// TIA Portal V17 export
// export: Created 2025-03-05T08:00:56.7108136Z, ExportSetting WithDefaults, DisplayName Totally Integrated Automation Portal, DisplayVersion V17 Update 8, DisplayName TIA Portal Openness, DisplayVersion V17 Update 8, DisplayName TIA Portal Version Control Interface, DisplayVersion V17, DisplayName SINAMICS Startdrive Advanced, DisplayVersion V17 SP2, DisplayName SINAMICS Startdrive G110M, G120, G120C, G120D, G120P, G115D, DisplayVersion V17 SP2, DisplayName SINAMICS Startdrive G130, G150, S120, S150, SINAMICS MV, S210, DisplayVersion V17 SP2, DisplayName STEP 7 Professional, DisplayVersion V17 Update 8, DisplayName SINUMERIK ONE STEP 7 Toolbox, DisplayVersion V17 Update 12, DisplayName SINUMERIK 840D sl STEP 7 Toolbox, DisplayVersion V17 Update 12, DisplayName STEP 7 Safety, DisplayVersion V17 Update 6, DisplayName WinCC Advanced, DisplayVersion V17 Update 8
FUNCTION "FC1502_PROTECTION_GAS" : Void   // FC1502, LAD
{ S7_Optimized_Access := 'TRUE' }
VERSION : 0.1
// stored: AutoNumber false, IsIECCheckEnabled false, SetENOAutomatically false, UDAEnableTagReadback false
   VAR_TEMP
      GAS_FLOW_TEMP_AUX : Real;
   END_VAR
BEGIN

REGION Network 1: PROTECTION GAS VALVE UNIT 01
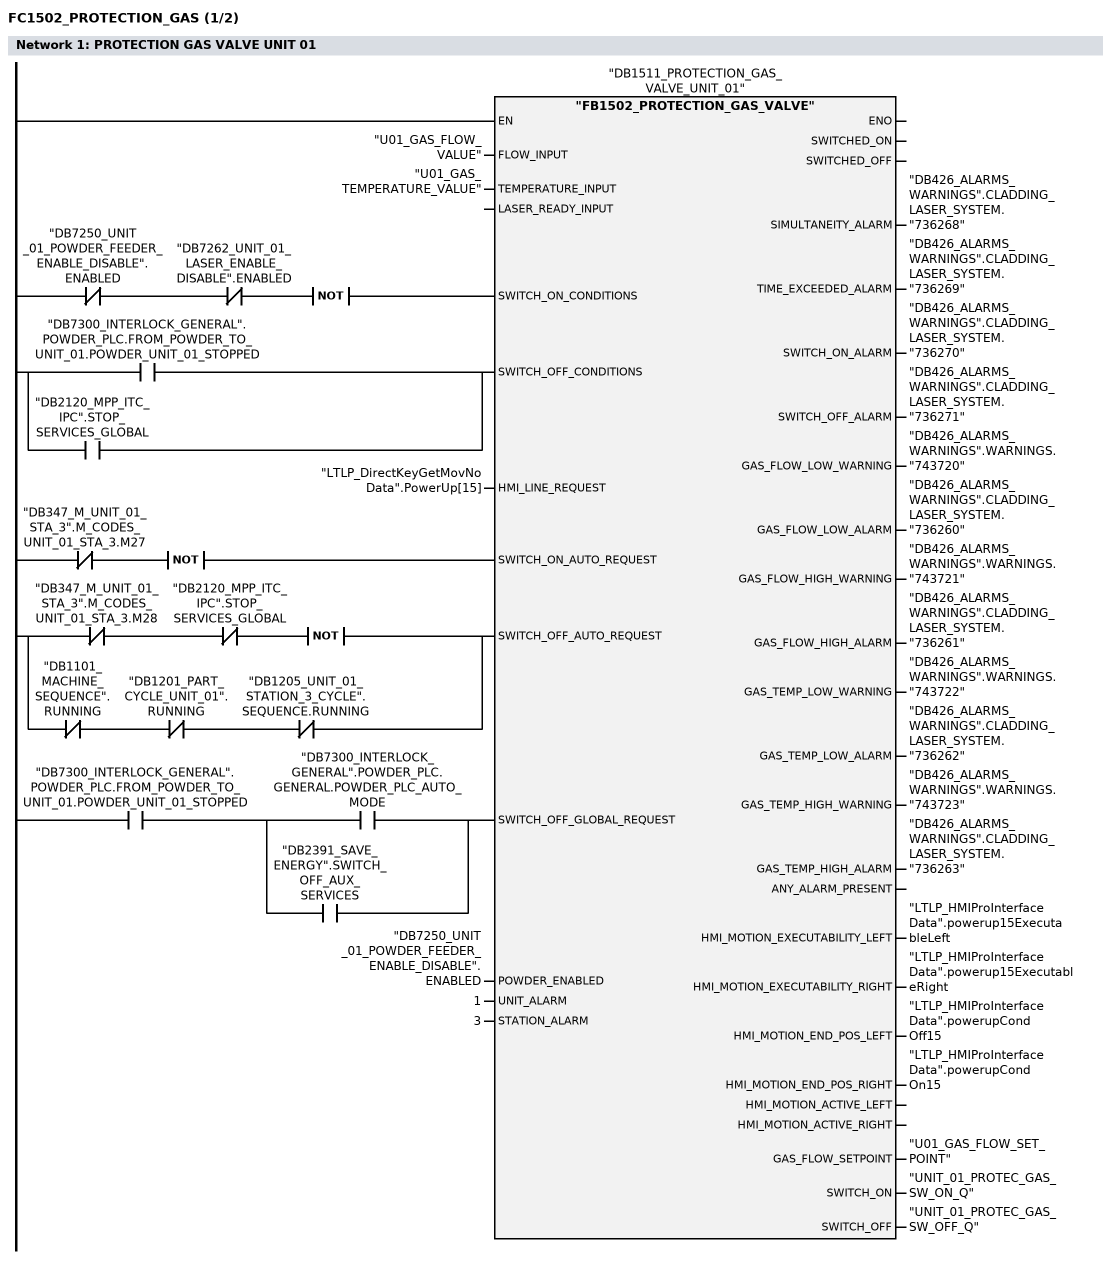
   RUNG wire#powerrail
      "DB1511_PROTECTION_GAS_VALVE_UNIT_01"(SWITCH_ON_CONDITIONS := wire#w1, SWITCH_OFF_CONDITIONS := wire#w2, SWITCH_ON_AUTO_REQUEST := wire#w3, SWITCH_OFF_AUTO_REQUEST := wire#w4, SWITCH_OFF_GLOBAL_REQUEST := wire#w6, FLOW_INPUT := "U01_GAS_FLOW_VALUE", TEMPERATURE_INPUT := "U01_GAS_TEMPERATURE_VALUE", LASER_READY_INPUT :=, HMI_LINE_REQUEST := "LTLP_DirectKeyGetMovNoData".PowerUp[15], POWDER_ENABLED := "DB7250_UNIT _01_POWDER_FEEDER_ENABLE_DISABLE".ENABLED, UNIT_ALARM := 1, STATION_ALARM := 3, SWITCHED_ON =>, SWITCHED_OFF =>, SIMULTANEITY_ALARM => "DB426_ALARMS_WARNINGS".CLADDING_LASER_SYSTEM."736268", TIME_EXCEEDED_ALARM => "DB426_ALARMS_WARNINGS".CLADDING_LASER_SYSTEM."736269", SWITCH_ON_ALARM => "DB426_ALARMS_WARNINGS".CLADDING_LASER_SYSTEM."736270", SWITCH_OFF_ALARM => "DB426_ALARMS_WARNINGS".CLADDING_LASER_SYSTEM."736271", GAS_FLOW_LOW_WARNING => "DB426_ALARMS_WARNINGS".WARNINGS."743720", GAS_FLOW_LOW_ALARM => "DB426_ALARMS_WARNINGS".CLADDING_LASER_SYSTEM."736260", GAS_FLOW_HIGH_WARNING => "DB426_ALARMS_WARNINGS".WARNINGS."743721", GAS_FLOW_HIGH_ALARM => "DB426_ALARMS_WARNINGS".CLADDING_LASER_SYSTEM."736261", GAS_TEMP_LOW_WARNING => "DB426_ALARMS_WARNINGS".WARNINGS."743722", GAS_TEMP_LOW_ALARM => "DB426_ALARMS_WARNINGS".CLADDING_LASER_SYSTEM."736262", GAS_TEMP_HIGH_WARNING => "DB426_ALARMS_WARNINGS".WARNINGS."743723", GAS_TEMP_HIGH_ALARM => "DB426_ALARMS_WARNINGS".CLADDING_LASER_SYSTEM."736263", ANY_ALARM_PRESENT =>, HMI_MOTION_EXECUTABILITY_LEFT => "LTLP_HMIProInterfaceData".powerup15ExecutableLeft, HMI_MOTION_EXECUTABILITY_RIGHT => "LTLP_HMIProInterfaceData".powerup15ExecutableRight, HMI_MOTION_END_POS_LEFT => "LTLP_HMIProInterfaceData".powerupCondOff15, HMI_MOTION_END_POS_RIGHT => "LTLP_HMIProInterfaceData".powerupCondOn15, HMI_MOTION_ACTIVE_LEFT =>, HMI_MOTION_ACTIVE_RIGHT =>, GAS_FLOW_SETPOINT => "U01_GAS_FLOW_SET_POINT", SWITCH_ON => "UNIT_01_PROTEC_GAS_SW_ON_Q", SWITCH_OFF => "UNIT_01_PROTEC_GAS_SW_OFF_Q")
   END_RUNG
   RUNG wire#powerrail
      I_Contact( "DB7250_UNIT _01_POWDER_FEEDER_ENABLE_DISABLE".ENABLED )
      I_Contact( "DB7262_UNIT_01_LASER_ENABLE_DISABLE".ENABLED )
      Not()
   END_RUNG wire#w1
   RUNG wire#powerrail
      Contact( "DB7300_INTERLOCK_GENERAL".POWDER_PLC.FROM_POWDER_TO_UNIT_01.POWDER_UNIT_01_STOPPED )
   END_RUNG wire#w2
   RUNG wire#powerrail
      Contact( "DB2120_MPP_ITC_IPC".STOP_SERVICES_GLOBAL )
   END_RUNG wire#w2
   RUNG wire#powerrail
      I_Contact( "DB347_M_UNIT_01_STA_3".M_CODES_UNIT_01_STA_3.M27 )
      Not()
   END_RUNG wire#w3
   RUNG wire#powerrail
      I_Contact( "DB347_M_UNIT_01_STA_3".M_CODES_UNIT_01_STA_3.M28 )
      I_Contact( "DB2120_MPP_ITC_IPC".STOP_SERVICES_GLOBAL )
      Not()
   END_RUNG wire#w4
   RUNG wire#powerrail
      I_Contact( "DB1101_MACHINE_SEQUENCE".RUNNING )
      I_Contact( "DB1201_PART_CYCLE_UNIT_01".RUNNING )
      I_Contact( "DB1205_UNIT_01_STATION_3_CYCLE".SEQUENCE.RUNNING )
   END_RUNG wire#w4
   RUNG wire#powerrail
      Contact( "DB7300_INTERLOCK_GENERAL".POWDER_PLC.FROM_POWDER_TO_UNIT_01.POWDER_UNIT_01_STOPPED )
      wire#w5
      Contact( "DB7300_INTERLOCK_GENERAL".POWDER_PLC.GENERAL.POWDER_PLC_AUTO_MODE )
   END_RUNG wire#w6
   RUNG wire#w5
      Contact( "DB2391_SAVE_ENERGY".SWITCH_OFF_AUX_SERVICES )
   END_RUNG wire#w6
   // the same network as SCL:
   "DB1511_PROTECTION_GAS_VALVE_UNIT_01"(FLOW_INPUT := "U01_GAS_FLOW_VALUE",   // "FB1502_PROTECTION_GAS_VALVE"
                           TEMPERATURE_INPUT := "U01_GAS_TEMPERATURE_VALUE",
                           SWITCH_ON_CONDITIONS := NOT (NOT "DB7250_UNIT _01_POWDER_FEEDER_ENABLE_DISABLE".ENABLED AND NOT "DB7262_UNIT_01_LASER_ENABLE_DISABLE".ENABLED),
                           SWITCH_OFF_CONDITIONS := "DB7300_INTERLOCK_GENERAL".POWDER_PLC.FROM_POWDER_TO_UNIT_01.POWDER_UNIT_01_STOPPED OR "DB2120_MPP_ITC_IPC".STOP_SERVICES_GLOBAL,
                           HMI_LINE_REQUEST := "LTLP_DirectKeyGetMovNoData".PowerUp[15],
                           SWITCH_ON_AUTO_REQUEST := NOT (NOT "DB347_M_UNIT_01_STA_3".M_CODES_UNIT_01_STA_3.M27),
                           SWITCH_OFF_AUTO_REQUEST := NOT (NOT "DB347_M_UNIT_01_STA_3".M_CODES_UNIT_01_STA_3.M28 AND NOT "DB2120_MPP_ITC_IPC".STOP_SERVICES_GLOBAL) OR (NOT "DB1101_MACHINE_SEQUENCE".RUNNING AND NOT "DB1201_PART_CYCLE_UNIT_01".RUNNING AND NOT "DB1205_UNIT_01_STATION_3_CYCLE".SEQUENCE.RUNNING),
                           SWITCH_OFF_GLOBAL_REQUEST := "DB7300_INTERLOCK_GENERAL".POWDER_PLC.FROM_POWDER_TO_UNIT_01.POWDER_UNIT_01_STOPPED AND ("DB7300_INTERLOCK_GENERAL".POWDER_PLC.GENERAL.POWDER_PLC_AUTO_MODE OR "DB2391_SAVE_ENERGY".SWITCH_OFF_AUX_SERVICES),
                           POWDER_ENABLED := "DB7250_UNIT _01_POWDER_FEEDER_ENABLE_DISABLE".ENABLED,
                           UNIT_ALARM := 1,
                           STATION_ALARM := 3,
                           SIMULTANEITY_ALARM => "DB426_ALARMS_WARNINGS".CLADDING_LASER_SYSTEM."736268",
                           TIME_EXCEEDED_ALARM => "DB426_ALARMS_WARNINGS".CLADDING_LASER_SYSTEM."736269",
                           SWITCH_ON_ALARM => "DB426_ALARMS_WARNINGS".CLADDING_LASER_SYSTEM."736270",
                           SWITCH_OFF_ALARM => "DB426_ALARMS_WARNINGS".CLADDING_LASER_SYSTEM."736271",
                           GAS_FLOW_LOW_WARNING => "DB426_ALARMS_WARNINGS".WARNINGS."743720",
                           GAS_FLOW_LOW_ALARM => "DB426_ALARMS_WARNINGS".CLADDING_LASER_SYSTEM."736260",
                           GAS_FLOW_HIGH_WARNING => "DB426_ALARMS_WARNINGS".WARNINGS."743721",
                           GAS_FLOW_HIGH_ALARM => "DB426_ALARMS_WARNINGS".CLADDING_LASER_SYSTEM."736261",
                           GAS_TEMP_LOW_WARNING => "DB426_ALARMS_WARNINGS".WARNINGS."743722",
                           GAS_TEMP_LOW_ALARM => "DB426_ALARMS_WARNINGS".CLADDING_LASER_SYSTEM."736262",
                           GAS_TEMP_HIGH_WARNING => "DB426_ALARMS_WARNINGS".WARNINGS."743723",
                           GAS_TEMP_HIGH_ALARM => "DB426_ALARMS_WARNINGS".CLADDING_LASER_SYSTEM."736263",
                           HMI_MOTION_EXECUTABILITY_LEFT => "LTLP_HMIProInterfaceData".powerup15ExecutableLeft,
                           HMI_MOTION_EXECUTABILITY_RIGHT => "LTLP_HMIProInterfaceData".powerup15ExecutableRight,
                           HMI_MOTION_END_POS_LEFT => "LTLP_HMIProInterfaceData".powerupCondOff15,
                           HMI_MOTION_END_POS_RIGHT => "LTLP_HMIProInterfaceData".powerupCondOn15,
                           GAS_FLOW_SETPOINT => "U01_GAS_FLOW_SET_POINT",
                           SWITCH_ON => "UNIT_01_PROTEC_GAS_SW_ON_Q",
                           SWITCH_OFF => "UNIT_01_PROTEC_GAS_SW_OFF_Q");
END_REGION

REGION Network 2: PROTECTION GAS VALVE UNIT 02
   // 2#0000_0001 OPTIONS 0 BIT 0 SWITCHED ON INPUT 1 OPTION
   // 2#0000_0010 OPTIONS 0 BIT 1 SWITCHED ON INPUT 2 OPTION
   // 2#0000_0100 OPTIONS 0 BIT 2 SWITCHED ON INPUT 3 OPTION
   // 2#0000_1000 OPTIONS 0 BIT 3 SWITCHED ON INPUT 4 OPTION
   // 2#0001_0000 OPTIONS 0 BIT 4 SWITCHED OFF NOT SWITCHED ON INPUT 1 OPTION
   // 2#0010_0000 OPTIONS 0 BIT 5 SPARE
   // 2#0100_0000 OPTIONS 0 BIT 6 SPARE
   // 2#1000_0000 OPTIONS 0 BIT 7 SPARE
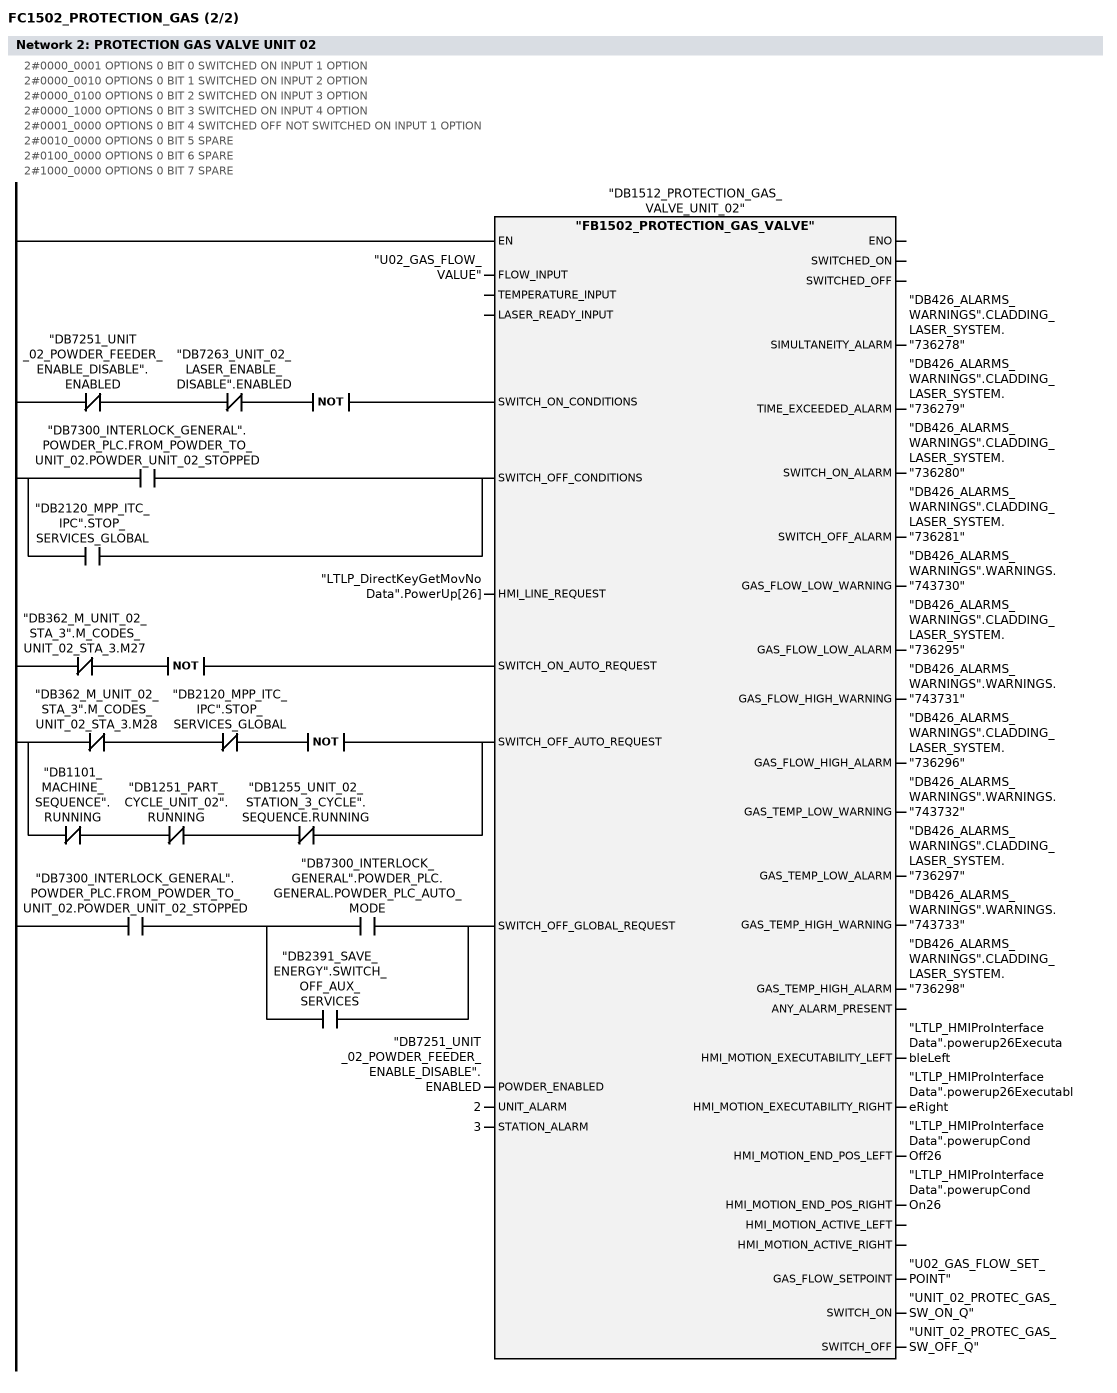
   RUNG wire#powerrail
      "DB1512_PROTECTION_GAS_VALVE_UNIT_02"(SWITCH_ON_CONDITIONS := wire#w1, SWITCH_OFF_CONDITIONS := wire#w2, SWITCH_ON_AUTO_REQUEST := wire#w3, SWITCH_OFF_AUTO_REQUEST := wire#w4, SWITCH_OFF_GLOBAL_REQUEST := wire#w6, FLOW_INPUT := "U02_GAS_FLOW_VALUE", TEMPERATURE_INPUT :=, LASER_READY_INPUT :=, HMI_LINE_REQUEST := "LTLP_DirectKeyGetMovNoData".PowerUp[26], POWDER_ENABLED := "DB7251_UNIT _02_POWDER_FEEDER_ENABLE_DISABLE".ENABLED, UNIT_ALARM := 2, STATION_ALARM := 3, SWITCHED_ON =>, SWITCHED_OFF =>, SIMULTANEITY_ALARM => "DB426_ALARMS_WARNINGS".CLADDING_LASER_SYSTEM."736278", TIME_EXCEEDED_ALARM => "DB426_ALARMS_WARNINGS".CLADDING_LASER_SYSTEM."736279", SWITCH_ON_ALARM => "DB426_ALARMS_WARNINGS".CLADDING_LASER_SYSTEM."736280", SWITCH_OFF_ALARM => "DB426_ALARMS_WARNINGS".CLADDING_LASER_SYSTEM."736281", GAS_FLOW_LOW_WARNING => "DB426_ALARMS_WARNINGS".WARNINGS."743730", GAS_FLOW_LOW_ALARM => "DB426_ALARMS_WARNINGS".CLADDING_LASER_SYSTEM."736295", GAS_FLOW_HIGH_WARNING => "DB426_ALARMS_WARNINGS".WARNINGS."743731", GAS_FLOW_HIGH_ALARM => "DB426_ALARMS_WARNINGS".CLADDING_LASER_SYSTEM."736296", GAS_TEMP_LOW_WARNING => "DB426_ALARMS_WARNINGS".WARNINGS."743732", GAS_TEMP_LOW_ALARM => "DB426_ALARMS_WARNINGS".CLADDING_LASER_SYSTEM."736297", GAS_TEMP_HIGH_WARNING => "DB426_ALARMS_WARNINGS".WARNINGS."743733", GAS_TEMP_HIGH_ALARM => "DB426_ALARMS_WARNINGS".CLADDING_LASER_SYSTEM."736298", ANY_ALARM_PRESENT =>, HMI_MOTION_EXECUTABILITY_LEFT => "LTLP_HMIProInterfaceData".powerup26ExecutableLeft, HMI_MOTION_EXECUTABILITY_RIGHT => "LTLP_HMIProInterfaceData".powerup26ExecutableRight, HMI_MOTION_END_POS_LEFT => "LTLP_HMIProInterfaceData".powerupCondOff26, HMI_MOTION_END_POS_RIGHT => "LTLP_HMIProInterfaceData".powerupCondOn26, HMI_MOTION_ACTIVE_LEFT =>, HMI_MOTION_ACTIVE_RIGHT =>, GAS_FLOW_SETPOINT => "U02_GAS_FLOW_SET_POINT", SWITCH_ON => "UNIT_02_PROTEC_GAS_SW_ON_Q", SWITCH_OFF => "UNIT_02_PROTEC_GAS_SW_OFF_Q")
   END_RUNG
   RUNG wire#powerrail
      I_Contact( "DB7251_UNIT _02_POWDER_FEEDER_ENABLE_DISABLE".ENABLED )
      I_Contact( "DB7263_UNIT_02_LASER_ENABLE_DISABLE".ENABLED )
      Not()
   END_RUNG wire#w1
   RUNG wire#powerrail
      Contact( "DB7300_INTERLOCK_GENERAL".POWDER_PLC.FROM_POWDER_TO_UNIT_02.POWDER_UNIT_02_STOPPED )
   END_RUNG wire#w2
   RUNG wire#powerrail
      Contact( "DB2120_MPP_ITC_IPC".STOP_SERVICES_GLOBAL )
   END_RUNG wire#w2
   RUNG wire#powerrail
      I_Contact( "DB362_M_UNIT_02_STA_3".M_CODES_UNIT_02_STA_3.M27 )
      Not()
   END_RUNG wire#w3
   RUNG wire#powerrail
      I_Contact( "DB362_M_UNIT_02_STA_3".M_CODES_UNIT_02_STA_3.M28 )
      I_Contact( "DB2120_MPP_ITC_IPC".STOP_SERVICES_GLOBAL )
      Not()
   END_RUNG wire#w4
   RUNG wire#powerrail
      I_Contact( "DB1101_MACHINE_SEQUENCE".RUNNING )
      I_Contact( "DB1251_PART_CYCLE_UNIT_02".RUNNING )
      I_Contact( "DB1255_UNIT_02_STATION_3_CYCLE".SEQUENCE.RUNNING )
   END_RUNG wire#w4
   RUNG wire#powerrail
      Contact( "DB7300_INTERLOCK_GENERAL".POWDER_PLC.FROM_POWDER_TO_UNIT_02.POWDER_UNIT_02_STOPPED )
      wire#w5
      Contact( "DB7300_INTERLOCK_GENERAL".POWDER_PLC.GENERAL.POWDER_PLC_AUTO_MODE )
   END_RUNG wire#w6
   RUNG wire#w5
      Contact( "DB2391_SAVE_ENERGY".SWITCH_OFF_AUX_SERVICES )
   END_RUNG wire#w6
   // the same network as SCL:
   "DB1512_PROTECTION_GAS_VALVE_UNIT_02"(FLOW_INPUT := "U02_GAS_FLOW_VALUE",   // "FB1502_PROTECTION_GAS_VALVE"
                           SWITCH_ON_CONDITIONS := NOT (NOT "DB7251_UNIT _02_POWDER_FEEDER_ENABLE_DISABLE".ENABLED AND NOT "DB7263_UNIT_02_LASER_ENABLE_DISABLE".ENABLED),
                           SWITCH_OFF_CONDITIONS := "DB7300_INTERLOCK_GENERAL".POWDER_PLC.FROM_POWDER_TO_UNIT_02.POWDER_UNIT_02_STOPPED OR "DB2120_MPP_ITC_IPC".STOP_SERVICES_GLOBAL,
                           HMI_LINE_REQUEST := "LTLP_DirectKeyGetMovNoData".PowerUp[26],
                           SWITCH_ON_AUTO_REQUEST := NOT (NOT "DB362_M_UNIT_02_STA_3".M_CODES_UNIT_02_STA_3.M27),
                           SWITCH_OFF_AUTO_REQUEST := NOT (NOT "DB362_M_UNIT_02_STA_3".M_CODES_UNIT_02_STA_3.M28 AND NOT "DB2120_MPP_ITC_IPC".STOP_SERVICES_GLOBAL) OR (NOT "DB1101_MACHINE_SEQUENCE".RUNNING AND NOT "DB1251_PART_CYCLE_UNIT_02".RUNNING AND NOT "DB1255_UNIT_02_STATION_3_CYCLE".SEQUENCE.RUNNING),
                           SWITCH_OFF_GLOBAL_REQUEST := "DB7300_INTERLOCK_GENERAL".POWDER_PLC.FROM_POWDER_TO_UNIT_02.POWDER_UNIT_02_STOPPED AND ("DB7300_INTERLOCK_GENERAL".POWDER_PLC.GENERAL.POWDER_PLC_AUTO_MODE OR "DB2391_SAVE_ENERGY".SWITCH_OFF_AUX_SERVICES),
                           POWDER_ENABLED := "DB7251_UNIT _02_POWDER_FEEDER_ENABLE_DISABLE".ENABLED,
                           UNIT_ALARM := 2,
                           STATION_ALARM := 3,
                           SIMULTANEITY_ALARM => "DB426_ALARMS_WARNINGS".CLADDING_LASER_SYSTEM."736278",
                           TIME_EXCEEDED_ALARM => "DB426_ALARMS_WARNINGS".CLADDING_LASER_SYSTEM."736279",
                           SWITCH_ON_ALARM => "DB426_ALARMS_WARNINGS".CLADDING_LASER_SYSTEM."736280",
                           SWITCH_OFF_ALARM => "DB426_ALARMS_WARNINGS".CLADDING_LASER_SYSTEM."736281",
                           GAS_FLOW_LOW_WARNING => "DB426_ALARMS_WARNINGS".WARNINGS."743730",
                           GAS_FLOW_LOW_ALARM => "DB426_ALARMS_WARNINGS".CLADDING_LASER_SYSTEM."736295",
                           GAS_FLOW_HIGH_WARNING => "DB426_ALARMS_WARNINGS".WARNINGS."743731",
                           GAS_FLOW_HIGH_ALARM => "DB426_ALARMS_WARNINGS".CLADDING_LASER_SYSTEM."736296",
                           GAS_TEMP_LOW_WARNING => "DB426_ALARMS_WARNINGS".WARNINGS."743732",
                           GAS_TEMP_LOW_ALARM => "DB426_ALARMS_WARNINGS".CLADDING_LASER_SYSTEM."736297",
                           GAS_TEMP_HIGH_WARNING => "DB426_ALARMS_WARNINGS".WARNINGS."743733",
                           GAS_TEMP_HIGH_ALARM => "DB426_ALARMS_WARNINGS".CLADDING_LASER_SYSTEM."736298",
                           HMI_MOTION_EXECUTABILITY_LEFT => "LTLP_HMIProInterfaceData".powerup26ExecutableLeft,
                           HMI_MOTION_EXECUTABILITY_RIGHT => "LTLP_HMIProInterfaceData".powerup26ExecutableRight,
                           HMI_MOTION_END_POS_LEFT => "LTLP_HMIProInterfaceData".powerupCondOff26,
                           HMI_MOTION_END_POS_RIGHT => "LTLP_HMIProInterfaceData".powerupCondOn26,
                           GAS_FLOW_SETPOINT => "U02_GAS_FLOW_SET_POINT",
                           SWITCH_ON => "UNIT_02_PROTEC_GAS_SW_ON_Q",
                           SWITCH_OFF => "UNIT_02_PROTEC_GAS_SW_OFF_Q");
END_REGION
END_FUNCTION
